// TIA Portal V16 export
// export: Created 2024-12-03T15:41:41.3900832Z, ExportSetting WithDefaults, DisplayName Totally Integrated Automation Portal, DisplayVersion V16 Update 6, DisplayName TIA Portal Version Control Interface, DisplayVersion V16 Update 2, DisplayName TIA Portal Openness, DisplayVersion V16 Update 6, DisplayName TIA Portal Teamcenter Gateway, DisplayVersion V16, DisplayName SINAMICS Startdrive Advanced, DisplayVersion V16 Update 5, DisplayName SINAMICS Startdrive G130, G150, S120, S150, SINAMICS MV, S210, DisplayVersion V16 Update 5, DisplayName SINAMICS Startdrive G110M, G120, G120C, G120D, G120P, G115D, DisplayVersion V16 Update 5, DisplayName STEP 7 Professional, DisplayVersion V16 Update 6, DisplayName STEP 7 Safety, DisplayVersion V16, DisplayName WinCC Advanced / Unified PC, DisplayVersion V16 Update 6
FUNCTION_BLOCK "StepperController_Encoder"   // FB59, SCL
{ S7_Optimized_Access := 'FALSE' }
VERSION : 0.1
// stored: AutoNumber true, IsIECCheckEnabled false, SetENOAutomatically false, UDAEnableTagReadback false
   VAR_INPUT
      I_StepNumber : DInt;
      I_NextStepNumber : DInt;
      I_ErrorStepNumber : DInt;
      I_TimeOutStepNumber : DInt;
      I_Condition : Bool;
      I_ErrorConditon : Bool;
      I_ConditionDistance : Real;
      I_TimeOutDistance : Real;
      I_ErrorDistance : Real;
      I_DeltaDistance : Real;
      I_IgnoreTimeOut : Bool;
      I_AccumulateConditionTIme : Bool;
      I_PauseTimeOut : Bool;
   END_VAR
   VAR_OUTPUT
      O_ConditionTrans : Bool;
      O_ErrorTrans : Bool;
      O_TimeTrans : Bool;
   END_VAR
   VAR_IN_OUT
      IO_StepNumber : DInt;
      IO_PrevStepNumber : DInt;
   END_VAR
   VAR
      ConditionTime { S7_SetPoint := 'True'} : "TON_Encoder_FB";
      TimeOutTime { S7_SetPoint := 'True'} : "TON_Encoder_FB";
      ErrorConditionTIme { S7_SetPoint := 'True'} : "TON_Encoder_FB";
   END_VAR
   VAR_TEMP
      T_SiemensBug : Bool;
   END_VAR
BEGIN
   //Reset flags
   #O_ConditionTrans := false;
   #O_ErrorTrans := false;
   #O_TimeTrans := FALSE;

   IF #I_StepNumber = #IO_StepNumber THEN

       REGION Check condition
           IF #I_ConditionDistance = 0.0 THEN
               IF #I_Condition THEN
                   "SetPrevStepNumber_FC"(I_Step:=#IO_StepNumber,
                                          IO_PrevStep:=#IO_PrevStepNumber);
                   #IO_StepNumber := #I_NextStepNumber;
                   #O_ConditionTrans := true;

               END_IF;
           ELSE
               #ConditionTime(I_Start := #I_Condition,
                              I_SetPoint:= #I_ConditionDistance,
                              I_DeltaDistance_mm:= #I_DeltaDistance);
               IF #ConditionTime.Q THEN
                   "SetPrevStepNumber_FC"(I_Step := #IO_StepNumber,
                                          IO_PrevStep := #IO_PrevStepNumber);
                   #IO_StepNumber := #I_NextStepNumber;
                   #O_ConditionTrans := true;

               END_IF;
           END_IF;

       END_REGION

       REGION Check Error conditon
           IF #I_ErrorDistance = 0.0 THEN
               IF #I_ErrorConditon THEN
                   "SetPrevStepNumber_FC"(I_Step := #IO_StepNumber,
                                          IO_PrevStep := #IO_PrevStepNumber);
                   #IO_StepNumber := #I_ErrorStepNumber;
                   #O_ErrorTrans := true;

               END_IF;
           ELSE
               #ErrorConditionTIme(I_Start := #I_ErrorConditon,
                                   I_SetPoint:= #I_ErrorDistance,
                                   I_DeltaDistance_mm := #I_DeltaDistance);
               IF #ErrorConditionTIme.Q THEN
                   "SetPrevStepNumber_FC"(I_Step := #IO_StepNumber,
                                          IO_PrevStep := #IO_PrevStepNumber);
                   #IO_StepNumber := #I_ErrorStepNumber;
                   #O_ErrorTrans := true;

               END_IF;
           END_IF;
       END_REGION

       REGION Check timeout

           #TimeOutTime(I_Start := #I_StepNumber = #IO_StepNumber AND NOT #I_IgnoreTimeOut AND NOT #I_PauseTimeOut ,
                        I_Reset:=NOT #I_AccumulateConditionTIme AND NOT (#I_StepNumber = #IO_StepNumber),
                        I_SetPoint:= #I_TimeOutDistance,
                        I_DeltaDistance_mm := #I_DeltaDistance,
                        I_Remanent := true,
                          Q=>#T_SiemensBug);

           IF #TimeOutTime.Q AND NOT #I_IgnoreTimeOut THEN
               "SetPrevStepNumber_FC"(I_Step := #IO_StepNumber,
                                      IO_PrevStep := #IO_PrevStepNumber);
               #IO_StepNumber := #I_TimeOutStepNumber;
               #O_TimeTrans := true;
               #TimeOutTime.DistanceMem := 0.0;

           END_IF;

       END_REGION
   ELSE
       #TimeOutTime.DistanceMem := 0.0;
       #ConditionTime.DistanceMem := 0.0;
       #ErrorConditionTIme.DistanceMem := 0.0;
       #O_ConditionTrans := FALSE;
       #O_ErrorTrans := FALSE;
       #O_TimeTrans := FALSE;
   END_IF;
END_FUNCTION_BLOCK
